PROGRAM MAIN
VAR
	// trigger command execution for Postman-Echo samples
	bGet, bGetPris, bPost, bPut, bHeaderAuth 	: BOOL;

	fbHttpClientSmartMeter			: FB_IotHttpClient :=(sHostName:='192.168.68.61',   //connectix_smartmeter.local
								  	bKeepAlive:=TRUE, tConnectionTimeout:=T#20S);
		
	fbHttpClientElpriset			: FB_IotHttpClient :=(sHostName:='elprisetjustnu.se',
	
								  	bKeepAlive:=TRUE, tConnectionTimeout:=T#5S);
									
	fbHttpClientSMHI			: FB_IotHttpClient :=(sHostName:='opendata-download-metfcst.smhi.se',
								  	bKeepAlive:=FALSE, tConnectionTimeout:=T#10S);

	fbHttpGet						: FB_HTTP_Get_SmartMeter;
	fbHttpGetElpriset				: FB_HTTP_Get_Elpris;
	fbHttpGetSMHI				: FB_HTTP_Get_SMHI;

	bGetSMHI: BOOL;
	samladataIntervall: TON;

	
	trigger: BOOL;
	loggadata: BOOL;
	raeknartid: TIME;
	systemtid: DT;
	nisse: INT;
	
//fbSystemTimeToFileTime: 	SYSTEMTIME_TO_FILETIME;

			 fbGetsytstemtime: GETSYSTEMTIME;
	 filetime: T_FILETIME;
	
	
	bGetSmartMeter: BOOL;
END_VAR


fbGetsytstemtime(timeLoDW=> filetime.dwLowDateTime, timeHiDW=> filetime.dwHighDateTime);
systemtid:= FILETIME_TO_DT(filetime);

//SmartMeter, hämta data en gång per 10sekunder

// init client parameters at startup
IF NOT fbHttpClientSmartMeter.bConfigured THEN 
	fbHttpClientSmartMeter.nHostPort:= 82;
END_IF

fbHttpClientSmartMeter.Execute();

samladataIntervall(IN:=trigger, PT:=  T#10S, Q=>bGetSmartMeter ,ET=> raeknartid);
IF samladataIntervall.Q THEN
	nisse:=nisse+1;			
	trigger:=FALSE;			
ELSE
		trigger:=TRUE;
END_IF

IF fbHttpClientSmartMeter.bConfigured THEN 
		fbHttpGet(bSend:=bGetSmartMeter, fbClient:=fbHttpClientSmartMeter);
END_IF




/////////////////////////////////////////////
//Elpriser 

// init client parameters at startup
IF NOT fbHttpClientElpriset.bConfigured THEN 
	//fbHttpClientElpriset.nHostPort:= 443;
	fbHttpClientElpriset.stTLS.sVersion:='tlsv1.3';
	

	
	
END_IF
IF fbHttpClientElpriset.bConfigured THEN 
	fbHttpGetElpriset(bSend:=bGetPris, fbClient:=fbHttpClientElpriset);
END_IF 

fbHttpClientElpriset.Execute();

/////////////////////////////////////////////
//SMHI

// init client parameters at startup
IF NOT fbHttpClientSMHI.bConfigured THEN 
	fbHttpClientSMHI.nHostPort:= 80;
	
	
END_IF
IF fbHttpClientSMHI.bConfigured THEN 
	fbHttpGetSMHI(bSend:=bGetSMHI, fbClient:=fbHttpClientSMHI);
END_IF 

fbHttpClientSMHI.Execute();

END_PROGRAM

(* stored: Version 1.1.0.1, ProductVersion 3.1.4024.12
   POU MAIN: Id {b37e2b32-48ef-44fd-8d39-b46780530972}, SpecialFunc None *)
